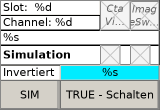
VISUALIZATION SimDO_Temp_Querry  // 160x110
VAR_INPUT	
	ITF_DO : ITF_DO;
END_VAR
    Frame (0,0 160x110)
        shows SimDO_Temp(ITF_DO := ITF_DO, IO_Ref_In := ITF_DO.proThisRef_DO)
END_VISUALIZATION

// 40 Visualizations/PFC VISU/PFC_SLOT
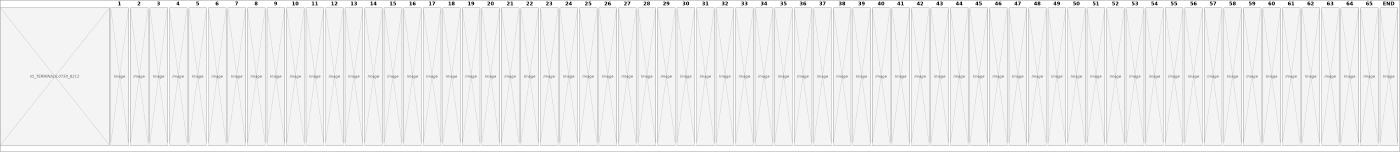
VISUALIZATION PFC_SLOT  // 3800x415
VAR_IN_OUT
    usiSelected :   USINT;	
END_VAR
    Rectangle (0,0 3800x415)
    Image (0,20 298x377), image: IO_TERMINALS.0750_8212
    Image (300,20 49x377), colour toggle: usiSelected = 1
        p84334746: fcGetModulImage(1)
        OnMouseDown: execute { usiSelected := 1; }
    Image (353,20 49x377), colour toggle: usiSelected = 2
        p84334746: fcGetModulImage(2)
        OnMouseDown: execute { usiSelected := 2; }
    Image (406,20 49x377), colour toggle: usiSelected = 3
        p84334746: fcGetModulImage(3)
        OnMouseDown: execute { usiSelected := 3; }
    Image (459,20 49x377), colour toggle: usiSelected = 4
        p84334746: fcGetModulImage(4)
        OnMouseDown: execute { usiSelected := 4; }
    Image (512,20 49x377), colour toggle: usiSelected = 5
        p84334746: fcGetModulImage(5)
        OnMouseDown: execute { usiSelected := 5; }
    Image (565,20 49x377), colour toggle: usiSelected = 6
        p84334746: fcGetModulImage(6)
        OnMouseDown: execute { usiSelected := 6; }
    Image (618,20 49x377), colour toggle: usiSelected = 7
        p84334746: fcGetModulImage(7)
        OnMouseDown: execute { usiSelected := 7; }
    Image (671,20 49x377), colour toggle: usiSelected = 8
        p84334746: fcGetModulImage(8)
        OnMouseDown: execute { usiSelected := 8; }
    Image (724,20 49x377), colour toggle: usiSelected = 9
        p84334746: fcGetModulImage(9)
        OnMouseDown: execute { usiSelected := 9; }
    Image (777,20 49x377), colour toggle: usiSelected = 10
        p84334746: fcGetModulImage(10)
        OnMouseDown: execute { usiSelected := 10; }
    Image (830,20 49x377), colour toggle: usiSelected = 11
        p84334746: fcGetModulImage(11)
        OnMouseDown: execute { usiSelected := 11; }
    Image (883,20 49x377), colour toggle: usiSelected = 12
        p84334746: fcGetModulImage(12)
        OnMouseDown: execute { usiSelected := 12; }
    Image (936,20 49x377), colour toggle: usiSelected = 13
        p84334746: fcGetModulImage(13)
        OnMouseDown: execute { usiSelected := 13; }
    Image (989,20 49x377), colour toggle: usiSelected = 14
        p84334746: fcGetModulImage(14)
        OnMouseDown: execute { usiSelected := 14; }
    Image (1042,20 49x377), colour toggle: usiSelected = 15
        p84334746: fcGetModulImage(15)
        OnMouseDown: execute { usiSelected := 15; }
    Image (1095,20 49x377), colour toggle: usiSelected = 16
        p84334746: fcGetModulImage(16)
        OnMouseDown: execute { usiSelected := 16; }
    Image (1148,20 49x377), colour toggle: usiSelected = 17
        p84334746: fcGetModulImage(17)
        OnMouseDown: execute { usiSelected := 17; }
    Image (1201,20 49x377), colour toggle: usiSelected = 18
        p84334746: fcGetModulImage(18)
        OnMouseDown: execute { usiSelected := 18; }
    Image (1254,20 49x377), colour toggle: usiSelected = 19
        p84334746: fcGetModulImage(19)
        OnMouseDown: execute { usiSelected := 19; }
    Image (1307,20 49x377), colour toggle: usiSelected = 20
        p84334746: fcGetModulImage(20)
        OnMouseDown: execute { usiSelected := 20; }
    Image (1413,20 49x377), colour toggle: usiSelected = 22
        p84334746: fcGetModulImage(22)
        OnMouseDown: execute { usiSelected := 22; }
    Image (1466,20 49x377), colour toggle: usiSelected = 23
        p84334746: fcGetModulImage(23)
        OnMouseDown: execute { usiSelected := 23; }
    Image (1519,20 49x377), colour toggle: usiSelected = 24
        p84334746: fcGetModulImage(24)
        OnMouseDown: execute { usiSelected := 24; }
    Image (1572,20 49x377), colour toggle: usiSelected = 25
        p84334746: fcGetModulImage(25)
        OnMouseDown: execute { usiSelected := 25; }
    Image (1625,20 49x377), colour toggle: usiSelected = 26
        p84334746: fcGetModulImage(26)
        OnMouseDown: execute { usiSelected := 26; }
    Image (1678,20 49x377), colour toggle: usiSelected = 27
        p84334746: fcGetModulImage(27)
        OnMouseDown: execute { usiSelected := 27; }
    Image (1731,20 49x377), colour toggle: usiSelected = 28
        p84334746: fcGetModulImage(28)
        OnMouseDown: execute { usiSelected := 28; }
    Image (1784,20 49x377), colour toggle: usiSelected = 29
        p84334746: fcGetModulImage(29)
        OnMouseDown: execute { usiSelected := 29; }
    Image (1837,20 49x377), colour toggle: usiSelected = 30
        p84334746: fcGetModulImage(30)
        OnMouseDown: execute { usiSelected := 30; }
    Image (1890,20 49x377), colour toggle: usiSelected = 31
        p84334746: fcGetModulImage(31)
        OnMouseDown: execute { usiSelected := 31; }
    Image (1943,20 49x377), colour toggle: usiSelected = 32
        p84334746: fcGetModulImage(32)
        OnMouseDown: execute { usiSelected := 32; }
    Image (1996,20 49x377), colour toggle: usiSelected = 33
        p84334746: fcGetModulImage(33)
        OnMouseDown: execute { usiSelected := 33; }
    Image (2049,20 49x377), colour toggle: usiSelected = 34
        p84334746: fcGetModulImage(34)
        OnMouseDown: execute { usiSelected := 34; }
    Image (2102,20 49x377), colour toggle: usiSelected = 35
        p84334746: fcGetModulImage(35)
        OnMouseDown: execute { usiSelected := 35; }
    Image (2155,20 49x377), colour toggle: usiSelected = 36
        p84334746: fcGetModulImage(36)
        OnMouseDown: execute { usiSelected := 36; }
    Image (2208,20 49x377), colour toggle: usiSelected = 37
        p84334746: fcGetModulImage(37)
        OnMouseDown: execute { usiSelected := 37; }
    Image (2261,20 49x377), colour toggle: usiSelected = 38
        p84334746: fcGetModulImage(38)
        OnMouseDown: execute { usiSelected := 38; }
    Image (2314,20 49x377), colour toggle: usiSelected = 39
        p84334746: fcGetModulImage(39)
        OnMouseDown: execute { usiSelected := 39; }
    Image (2367,20 49x377), colour toggle: usiSelected = 40
        p84334746: fcGetModulImage(40)
        OnMouseDown: execute { usiSelected := 40; }
    Image (2420,20 49x377), colour toggle: usiSelected = 41
        p84334746: fcGetModulImage(41)
        OnMouseDown: execute { usiSelected := 41; }
    Image (2473,20 49x377), colour toggle: usiSelected = 42
        p84334746: fcGetModulImage(42)
        OnMouseDown: execute { usiSelected := 42; }
    Image (2526,20 49x377), colour toggle: usiSelected = 43
        p84334746: fcGetModulImage(43)
        OnMouseDown: execute { usiSelected := 43; }
    Image (2579,20 49x377), colour toggle: usiSelected = 44
        p84334746: fcGetModulImage(44)
        OnMouseDown: execute { usiSelected := 44; }
    Image (2632,20 49x377), colour toggle: usiSelected = 45
        p84334746: fcGetModulImage(45)
        OnMouseDown: execute { usiSelected := 45; }
    Image (2685,20 49x377), colour toggle: usiSelected = 46
        p84334746: fcGetModulImage(46)
        OnMouseDown: execute { usiSelected := 46; }
    Image (2738,20 49x377), colour toggle: usiSelected = 47
        p84334746: fcGetModulImage(47)
        OnMouseDown: execute { usiSelected := 47; }
    Image (2791,20 49x377), colour toggle: usiSelected = 48
        p84334746: fcGetModulImage(48)
        OnMouseDown: execute { usiSelected := 48; }
    Image (2844,20 49x377), colour toggle: usiSelected = 49
        p84334746: fcGetModulImage(49)
        OnMouseDown: execute { usiSelected := 49; }
    Image (2897,20 49x377), colour toggle: usiSelected = 50
        p84334746: fcGetModulImage(50)
        OnMouseDown: execute { usiSelected := 50; }
    Image (2950,20 49x377), colour toggle: usiSelected = 51
        p84334746: fcGetModulImage(51)
        OnMouseDown: execute { usiSelected := 51; }
    Image (3003,20 49x377), colour toggle: usiSelected = 52
        p84334746: fcGetModulImage(52)
        OnMouseDown: execute { usiSelected := 52; }
    Image (3056,20 49x377), colour toggle: usiSelected = 53
        p84334746: fcGetModulImage(53)
        OnMouseDown: execute { usiSelected := 53; }
    Image (3109,20 49x377), colour toggle: usiSelected = 54
        p84334746: fcGetModulImage(54)
        OnMouseDown: execute { usiSelected := 54; }
    Image (3162,20 49x377), colour toggle: usiSelected = 55
        p84334746: fcGetModulImage(55)
        OnMouseDown: execute { usiSelected := 55; }
    Image (3215,20 49x377), colour toggle: usiSelected = 56
        p84334746: fcGetModulImage(56)
        OnMouseDown: execute { usiSelected := 56; }
    Image (3268,20 49x377), colour toggle: usiSelected = 57
        p84334746: fcGetModulImage(57)
        OnMouseDown: execute { usiSelected := 57; }
    Image (3321,20 49x377), colour toggle: usiSelected = 58
        p84334746: fcGetModulImage(58)
        OnMouseDown: execute { usiSelected := 58; }
    Image (3374,20 49x377), colour toggle: usiSelected = 59
        p84334746: fcGetModulImage(59)
        OnMouseDown: execute { usiSelected := 59; }
    Image (3427,20 49x377), colour toggle: usiSelected = 60
        p84334746: fcGetModulImage(60)
        OnMouseDown: execute { usiSelected := 60; }
    Image (1360,20 49x377), colour toggle: usiSelected = 21
        p84334746: fcGetModulImage(21)
        OnMouseDown: execute { usiSelected := 21; }
    Image (3692,20 49x377), colour toggle: usiSelected = 65
        p84334746: fcGetModulImage(65)
        OnMouseDown: execute { usiSelected := 65; }
    Image (3480,20 49x377), colour toggle: usiSelected = 61
        p84334746: fcGetModulImage(61)
        OnMouseDown: execute { usiSelected := 61; }
    Image (3533,20 49x377), colour toggle: usiSelected = 62
        p84334746: fcGetModulImage(62)
        OnMouseDown: execute { usiSelected := 62; }
    Image (3586,20 49x377), colour toggle: usiSelected = 63
        p84334746: fcGetModulImage(63)
        OnMouseDown: execute { usiSelected := 63; }
    Image (3639,20 49x377), colour toggle: usiSelected = 64
        p84334746: fcGetModulImage(64)
        OnMouseDown: execute { usiSelected := 64; }
    Image (3745,20 49x377)
        p84334746: fcGetModulImage(66)
    Label (300,0 49x20), "1"
    Label (353,0 49x20), "2"
    Label (406,0 49x20), "3"
    Label (565,0 49x20), "6"
    Label (459,0 49x20), "4"
    Label (512,0 49x20), "5"
    Label (883,0 49x20), "12"
    Label (618,0 49x20), "7"
    Label (671,0 49x20), "8"
    Label (724,0 49x20), "9"
    Label (777,0 49x20), "10"
    Label (830,0 49x20), "11"
    Label (1201,0 49x20), "18"
    Label (936,0 49x20), "13"
    Label (989,0 49x20), "14"
    Label (1042,0 49x20), "15"
    Label (1095,0 49x20), "16"
    Label (1148,0 49x20), "17"
    Label (1254,0 49x20), "19"
    Label (1307,0 49x20), "20"
    Label (1360,0 49x20), "21"
    Label (1519,0 49x20), "24"
    Label (1413,0 49x20), "22"
    Label (1466,0 49x20), "23"
    Label (1837,0 49x20), "30"
    Label (1572,0 49x20), "25"
    Label (1625,0 49x20), "26"
    Label (1678,0 49x20), "27"
    Label (1731,0 49x20), "28"
    Label (1784,0 49x20), "29"
    Label (2155,0 49x20), "36"
    Label (1890,0 49x20), "31"
    Label (1943,0 49x20), "32"
    Label (1996,0 49x20), "33"
    Label (2049,0 49x20), "34"
    Label (2102,0 49x20), "35"
    Label (2208,0 49x20), "37"
    Label (2261,0 49x20), "38"
    Label (2314,0 49x20), "39"
    Label (2473,0 49x20), "42"
    Label (2367,0 49x20), "40"
    Label (2420,0 49x20), "41"
    Label (2791,0 49x20), "48"
    Label (2526,0 49x20), "43"
    Label (2579,0 49x20), "44"
    Label (2632,0 49x20), "45"
    Label (2685,0 49x20), "46"
    Label (2738,0 49x20), "47"
    Label (3109,0 49x20), "54"
    Label (2844,0 49x20), "49"
    Label (2897,0 49x20), "50"
    Label (2950,0 49x20), "51"
    Label (3003,0 49x20), "52"
    Label (3056,0 49x20), "53"
    Label (3162,0 49x20), "55"
    Label (3215,0 49x20), "56"
    Label (3268,0 49x20), "57"
    Label (3427,0 49x20), "60"
    Label (3321,0 49x20), "58"
    Label (3374,0 49x20), "59"
    Label (3745,0 49x20), "END"
    Label (3480,0 49x20), "61"
    Label (3533,0 49x20), "62"
    Label (3586,0 49x20), "63"
    Label (3639,0 49x20), "64"
    Label (3692,0 49x20), "65"
END_VISUALIZATION

// 40 Visualizations/PFC VISU/IO_Manager_Base
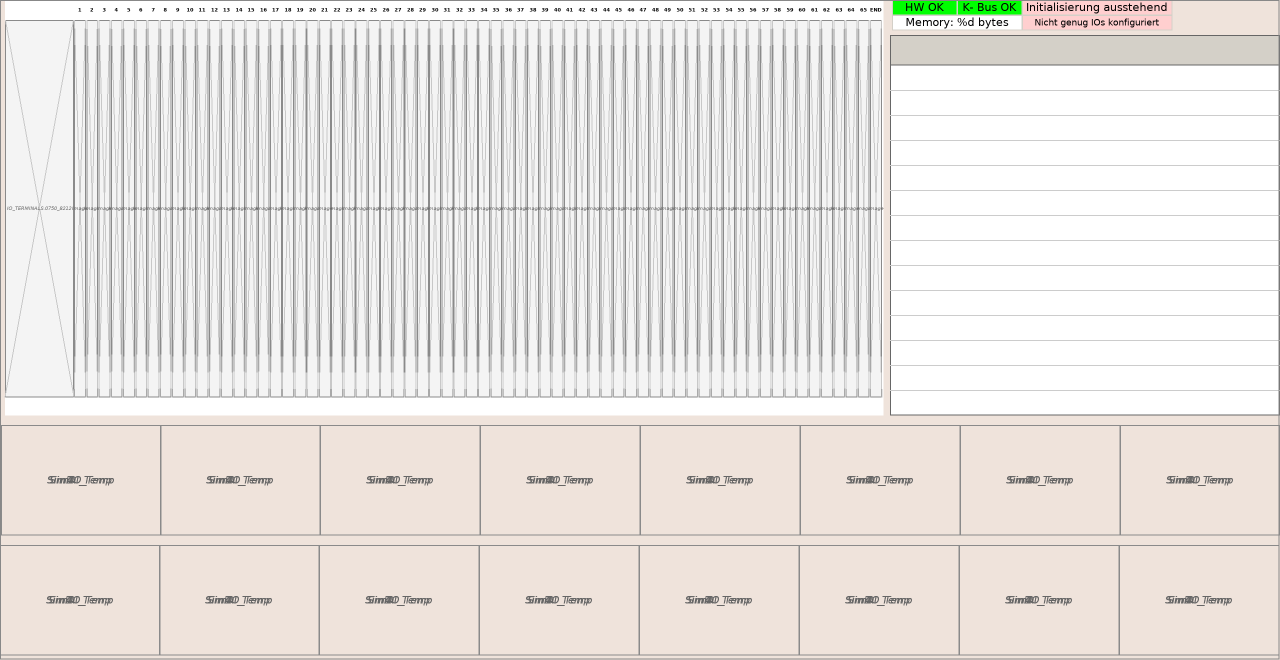
VISUALIZATION IO_Manager_Base  // 1280x660
VAR_INPUT
    ayIOs			    :	ARRAY [1..Parameter.MAX_NUM_OF_IOS] OF ITF_IO;
	xErrNotEnoughIOs	:	BOOL;
	xIoInitDone		    : 	BOOL;
	xKbusErrHW		    :	BOOL;
	xKbusErrSW		    : 	BOOL;
	iMax				:	INT;
	udiNeededMemSize	: 	UDINT;
END_VAR
VAR
    iZeile              :   INT;
    usiSelected         :   USINT;	
    fbPfcVisuHelp       :   fbPfcVisuHelp;
END_VAR
    Frame (5,0 878x415), invisible if: fbPfcVisuHelp.getSizeOfFrame(This^.GEN_Instance_PFC_SLOT_0.GetSize())
        shows PFC_SLOT(usiSelected := usiSelected)
        p3549101943: fbPfcVisuHelp.proScrollBar
    Frame (1,425 160x110), invisible if: fbPfcVisuHelp.metNotShowChannel(1)
        shows Simulation(ITF_IO := ayIOs[fbPfcVisuHelp.metGetSlotIos(ayIOs:= ayIOs,iMax:= iMax,iChannel:= 1,iZeile:= iZeile,usiSlot:= usiSelected)])
    Frame (160,425 160x110), invisible if: fbPfcVisuHelp.metNotShowChannel(2)
        shows Simulation(ITF_IO := ayIOs[fbPfcVisuHelp.metGetSlotIos(ayIOs:= ayIOs,iMax:= iMax,iChannel:= 2,iZeile:= iZeile,usiSlot:= usiSelected)])
    Frame (320,425 160x110), invisible if: fbPfcVisuHelp.metNotShowChannel(3)
        shows Simulation(ITF_IO := ayIOs[fbPfcVisuHelp.metGetSlotIos(ayIOs:= ayIOs,iMax:= iMax,iChannel:= 3,iZeile:= iZeile,usiSlot:= usiSelected)])
    Frame (480,425 160x110), invisible if: fbPfcVisuHelp.metNotShowChannel(4)
        shows Simulation(ITF_IO := ayIOs[fbPfcVisuHelp.metGetSlotIos(ayIOs:= ayIOs,iMax:= iMax,iChannel:= 4,iZeile:= iZeile,usiSlot:= usiSelected)])
    Frame (0,545 160x110), invisible if: fbPfcVisuHelp.metNotShowChannel(9)
        shows Simulation(ITF_IO := ayIOs[fbPfcVisuHelp.metGetSlotIos(ayIOs:= ayIOs,iMax:= iMax,iChannel:= 9,iZeile:= iZeile,usiSlot:= usiSelected)])
    Frame (892,0 280x30)
        shows IO_ManagerBusInfo(xErrNotEnoughIOs := xErrNotEnoughIOs, xIoInitDone := xIoInitDone, xKbusErrHW := xKbusErrHW, xKbusErrSW := xKbusErrSW, udiNeededMemSize := udiNeededMemSize)
    Frame (159,545 160x110), invisible if: fbPfcVisuHelp.metNotShowChannel(10)
        shows Simulation(ITF_IO := ayIOs[fbPfcVisuHelp.metGetSlotIos(ayIOs:= ayIOs,iMax:= iMax,iChannel:= 10,iZeile:= iZeile,usiSlot:= usiSelected)])
    Frame (319,545 160x110), invisible if: fbPfcVisuHelp.metNotShowChannel(11)
        shows Simulation(ITF_IO := ayIOs[fbPfcVisuHelp.metGetSlotIos(ayIOs:= ayIOs,iMax:= iMax,iChannel:= 11,iZeile:= iZeile,usiSlot:= usiSelected)])
    Frame (479,545 160x110), invisible if: fbPfcVisuHelp.metNotShowChannel(12)
        shows Simulation(ITF_IO := ayIOs[fbPfcVisuHelp.metGetSlotIos(ayIOs:= ayIOs,iMax:= iMax,iChannel:= 12,iZeile:= iZeile,usiSlot:= usiSelected)])
    Frame (1120,425 160x110), invisible if: fbPfcVisuHelp.metNotShowChannel(8)
        shows Simulation(ITF_IO := ayIOs[fbPfcVisuHelp.metGetSlotIos(ayIOs:= ayIOs,iMax:= iMax,iChannel:= 8,iZeile:= iZeile,usiSlot:= usiSelected)])
    Frame (640,425 160x110), invisible if: fbPfcVisuHelp.metNotShowChannel(5)
        shows Simulation(ITF_IO := ayIOs[fbPfcVisuHelp.metGetSlotIos(ayIOs:= ayIOs,iMax:= iMax,iChannel:= 5,iZeile:= iZeile,usiSlot:= usiSelected)])
    Frame (800,425 160x110), invisible if: fbPfcVisuHelp.metNotShowChannel(6)
        shows Simulation(ITF_IO := ayIOs[fbPfcVisuHelp.metGetSlotIos(ayIOs:= ayIOs,iMax:= iMax,iChannel:= 6,iZeile:= iZeile,usiSlot:= usiSelected)])
    Frame (960,425 160x110), invisible if: fbPfcVisuHelp.metNotShowChannel(7)
        shows Simulation(ITF_IO := ayIOs[fbPfcVisuHelp.metGetSlotIos(ayIOs:= ayIOs,iMax:= iMax,iChannel:= 7,iZeile:= iZeile,usiSlot:= usiSelected)])
    Frame (639,545 160x110), invisible if: fbPfcVisuHelp.metNotShowChannel(13)
        shows Simulation(ITF_IO := ayIOs[fbPfcVisuHelp.metGetSlotIos(ayIOs:= ayIOs,iMax:= iMax,iChannel:= 13,iZeile:= iZeile,usiSlot:= usiSelected)])
    Frame (799,545 160x110), invisible if: fbPfcVisuHelp.metNotShowChannel(14)
        shows Simulation(ITF_IO := ayIOs[fbPfcVisuHelp.metGetSlotIos(ayIOs:= ayIOs,iMax:= iMax,iChannel:= 14,iZeile:= iZeile,usiSlot:= usiSelected)])
    Frame (959,545 160x110), invisible if: fbPfcVisuHelp.metNotShowChannel(15)
        shows Simulation(ITF_IO := ayIOs[fbPfcVisuHelp.metGetSlotIos(ayIOs:= ayIOs,iMax:= iMax,iChannel:= 15,iZeile:= iZeile,usiSlot:= usiSelected)])
    Frame (1119,545 160x110), invisible if: fbPfcVisuHelp.metNotShowChannel(16)
        shows Simulation(ITF_IO := ayIOs[fbPfcVisuHelp.metGetSlotIos(ayIOs:= ayIOs,iMax:= iMax,iChannel:= 16,iZeile:= iZeile,usiSlot:= usiSelected)])
    Table (890,35 390x380), data array: ayIOs
        p1014161805: Parameter.MAX_NUM_OF_IOS - 1 + INT#1
        p1128707560: iMax
        p1137915858: iZeile
        p2232123230: Slot
        p2685023577: ayIOs[INDEX].proSlot
        p511219082: Channel
        p3312258591: ayIOs[INDEX].proChannel
        p4242324053: ayIOs[INDEX].proChannelAdress
        p1755163831: Modul Type
        p1791247317: ayIOs[INDEX].proModuleType
        p262371475: ayIOs[INDEX].proOkVisu
        p4008173056: ayIOs[INDEX].proSimVisu
        p1739542657: ayIOs[INDEX].P_scfbIO_fbxSimulationLock
        p516019884: ayIOs[INDEX].proOK
        p2243050616: ayIOs[INDEX].proKbusOk
        p4088588272: ayIOs[INDEX].proIsHand
        p1757482276: ayIOs[INDEX].P_scfbIO_Simulation
        p505689113: Value
        p2340480326: ayIOs[INDEX].proPhysikalValueVisu
END_VISUALIZATION

// 40 Visualizations/PFC VISU/IO_Manager_Sync
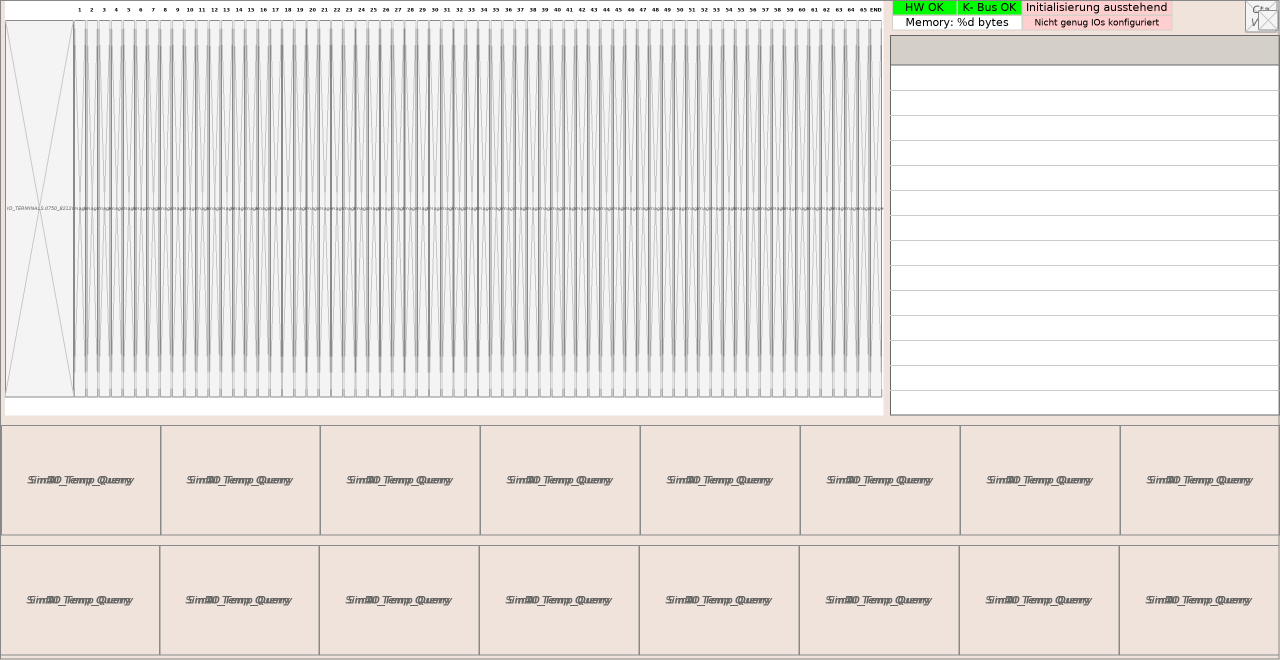
VISUALIZATION IO_Manager_Sync  // 1280x660
VAR_INPUT
	ITF_IO_Manager_Visu : ITF_IO_Manager_Visu;
END_VAR
    Frame (0,0 1280x660), invisible if: NOT __QUERYINTERFACE(ITF_IO_Manager_Visu,ITF_IO_Manager_Visu)
        shows IO_Manager_Base(ayIOs := ITF_IO_Manager_Visu.proAyIOs, xErrNotEnoughIOs := ITF_IO_Manager_Visu.proErrNotEnoughIOs, xIoInitDone := ITF_IO_Manager_Visu.proIoInitDone, xKbusErrHW := ITF_IO_Manager_Visu.proKbusErrHW, xKbusErrSW := ITF_IO_Manager_Visu.proKbusErrSW, iMax := ITF_IO_Manager_Visu.proMaxIO, udiNeededMemSize := ITF_IO_Manager_Visu.proNeededMemSize)
    Image (1245,0 32x32), invisible if: NOt ITF_IO_Manager_Visu.proAllowSim, input disabled if: NOt ITF_IO_Manager_Visu.proAllowSim, image: CtaVisSymbols.ImagePool.dip-switch
        OnMouseClick: execute { ITF_IO_Manager_Visu.proSimOn := NOT ITF_IO_Manager_Visu.proSimOn; }
    Image (1258,10 20x20), invisible if: NOT ITF_IO_Manager_Visu.proSimOn, image: CtaVisSymbols.ImagePool.front_hand_Yellow
END_VISUALIZATION

// 40 Visualizations/PFC VISU/IO_Manager_View
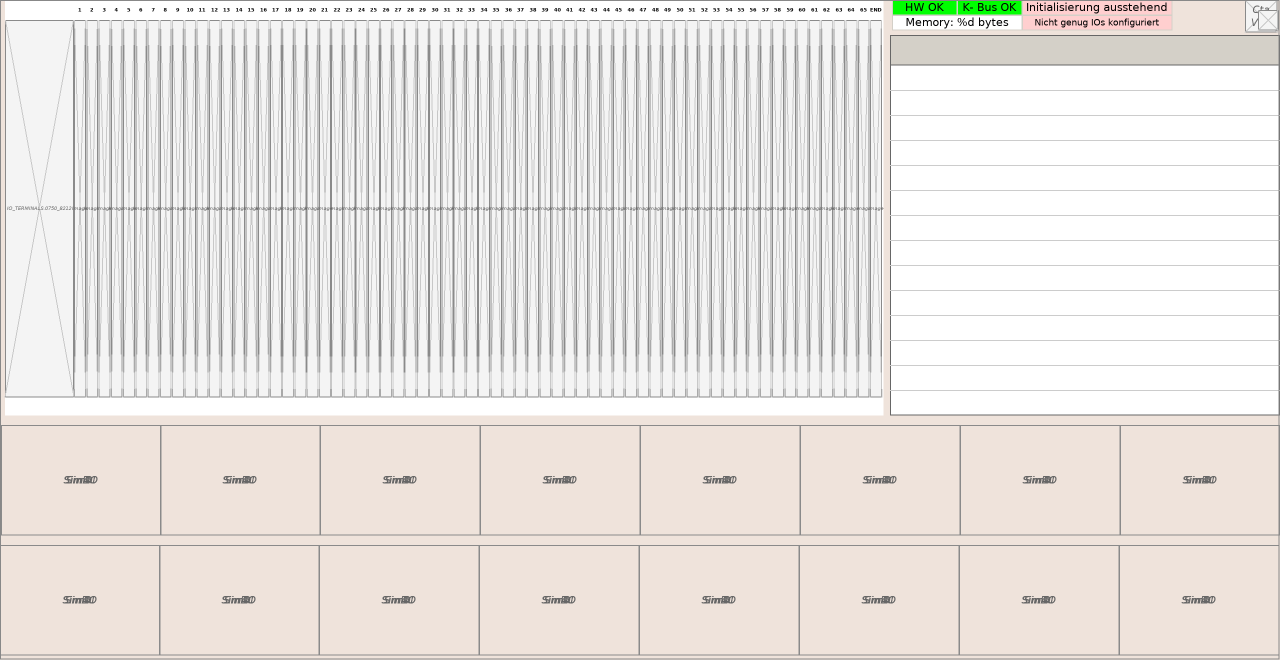
VISUALIZATION IO_Manager_View  // 1280x660
    Frame (0,0 1280x660)
        shows IO_Manager_Sync(ITF_IO_Manager_Visu := GVL_IO.fbIO_Manager)
END_VISUALIZATION

// 40 Visualizations/Simulation/DIA_IO_CONFIG
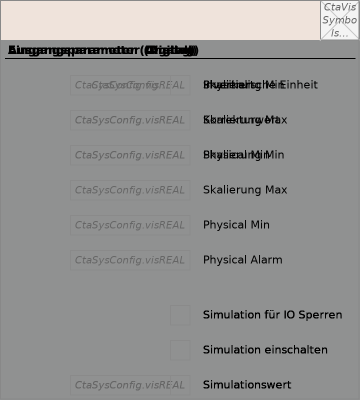
VISUALIZATION DIA_IO_CONFIG  // 360x400
VAR_INPUT
    ITF_IO_IN 	: 	ITF_IO;
END_VAR
    Rectangle (0,0 360x400)
    Frame (0,40 360x360)
        shows VIS_IO_PARAMETER_BASE(ITF_IO_IN := ITF_IO_IN)
    Image (320,0 40x40), image: CtaVisSymbols.ImagePool.close_solo_black
        OnMouseClick:  Dialog=DIA_IO_CONFIG, Result=OK, NumpadKeypadSet=True
END_VISUALIZATION

(* text list txtModulType (id | default)
  Unknown | Unbekannt
  Digital_IN | Digital IN
  Digital_OUT | Digital OUT
  DC_0_10V_IN | DC 0-10V IN
  DC_0_10V_OUT | DC 0-10V OUT
  DC_4_20mA_IN | DC 4-20mA IN
  DC_4_20mA_OUT | DC 4-20mA Out
  ohm | Ohm
   |  *)

(* text list txtWarning (id | default)
  91 | IO Handeingriff
   |  *)

(* text list txtError (id | default)
  91 | K-Bus Error Reboot notwendig
  92 | Modulkonfigurations Fehler. Module stimmen nicht mit Software überein
   |  *)

(* text list txtPhysicalUnit (id | default)
  0 | NaN
  1 | Digital In
  2 | Digital Out
  3 | 0 - 10 V
  4 | 4 - 20 mA
  5 | 0 - 10 V
  6 | 4 - 20 mA
  7 | °C
  8 | 
  9 | 0 - 20 mA
   |  *)
